FUNCTION Convert_TIME_TO_INT : Hresult
VAR_INPUT
	in : TIME;
	out : REFERENCE TO INT;
END_VAR
VAR
	converted : INT;
END_VAR

converted := TIME_TO_INT(in);

IF (INT_TO_TIME(converted) <> in) THEN
	Convert_TIME_TO_INT := INCOMPATIBLE;
	RETURN;
END_IF

out := converted;

END_FUNCTION

(* stored: Version 1.1.0.1, ProductVersion 3.1.4024.12
   POU Convert_TIME_TO_INT: Id {ee185f76-6201-416c-83e7-619f85ba77e5}, SpecialFunc None *)
